TYPE Kickout_IO_typ:
STRUCT
	Inputs	:  Kickout_Inputs_typ;
	Outputs	: Kickout_Outputs_typ;
END_STRUCT
END_TYPE

(* stored: Version 1.1.0.1, ProductVersion 3.1.4024.12
   DUT Kickout_IO_typ: Id {de8c3c0c-5df9-0c7d-2737-6c5930d793e0} *)
